SUBAPPLICATION GreenWhiteBackground_Function (* Subapplication Type *)
  (* Standard: 61499-2 *)
  (* Version 1.0, 2023-02-06, franz *)
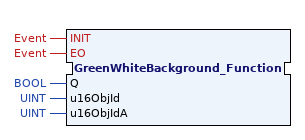
  EVENT_INPUT
    INIT;
    EO;
  END_EVENT
  VAR_INPUT
    Q : BOOL;
    u16ObjId : UINT;
    u16ObjIdA : UINT;
  END_VAR
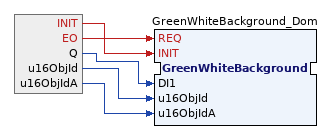
  SUBAPPS
    GreenWhiteBackground_Dom : GreenWhiteBackground;
  END_SUBAPPS
  EVENT_CONNECTIONS
    EO TO GreenWhiteBackground_Dom.REQ;
    INIT TO GreenWhiteBackground_Dom.INIT;
  END_CONNECTIONS
  DATA_CONNECTIONS
    Q TO GreenWhiteBackground_Dom.DI1;
    u16ObjId TO GreenWhiteBackground_Dom.u16ObjId;
    u16ObjIdA TO GreenWhiteBackground_Dom.u16ObjIdA;
  END_CONNECTIONS
END_SUBAPPLICATION
